{attribute 'GeneratedUsingTerminal: EP3744-0041-0016'}
{attribute addProperty BoxType "EP3744-0041-0016"}
{attribute addProperty Description "EP3744-0041 5Ch. Absolute Pressure 6Ch. Dig. Input 10us 2Ch. Dig. Output 24V 0,5A M8"}
{attribute addProperty Physics "YY"}
{attribute addProperty Id "DIG_InputsAT %I*DIG_Inputs_697E0EF26AI_Inputs_Channel_1AT %I*AI_Inputs_Channel_4521310411AI_Inputs_Channel_2AT %I*AI_Inputs_Channel_4521310411AI_Inputs_Channel_3AT %I*AI_Inputs_Channel_4521310411AI_Inputs_Channel_4AT %I*AI_Inputs_Channel_4521310411DEV_Inputs_DeviceAT %I*DEV_Inputs_Device_5F4E175E5DIG_OutputsAT %Q*DIG_Outputs_DE230DD52DEV_Outputs_DeviceAT %Q*DEV_Outputs_Device_59FFD2471WcStateAT %I*WcState_9091E0EB2InfoDataAT %I*InfoData_32EB74EA10"}
{attribute addProperty CRC "828150484"}
{attribute addProperty Size "70"}
TYPE EP3744_315C92D4 EXTENDS EtcSlaveBoxBase_77A0E4A7 :
STRUCT
	{attribute addProperty Name "DIG_Inputs"}
	DIG_Inputs : DIG_Inputs_697E0EF2;
	{attribute addProperty Name "AI_Inputs_Channel_1"}
	AI_Inputs_Channel_1 : AI_Inputs_Channel_45213104;
	{attribute addProperty Name "AI_Inputs_Channel_2"}
	AI_Inputs_Channel_2 : AI_Inputs_Channel_45213104;
	{attribute addProperty Name "AI_Inputs_Channel_3"}
	AI_Inputs_Channel_3 : AI_Inputs_Channel_45213104;
	{attribute addProperty Name "AI_Inputs_Channel_4"}
	AI_Inputs_Channel_4 : AI_Inputs_Channel_45213104;
	{attribute addProperty Name "DEV_Inputs_Device"}
	DEV_Inputs_Device : DEV_Inputs_Device_5F4E175E;
	{attribute addProperty Name "DIG_Outputs"}
	DIG_Outputs : DIG_Outputs_DE230DD5;
	{attribute addProperty Name "DEV_Outputs_Device"}
	DEV_Outputs_Device : DEV_Outputs_Device_59FFD247;
	{attribute addProperty Name "WcState"}
	WcState : WcState_9091E0EB;
	{attribute addProperty Name "InfoData"}
	InfoData : InfoData_32EB74EA;
END_STRUCT
END_TYPE

(* stored: Version 1.2.0.0, ProductVersion 3.1.4024.9
   DUT EP3744_315C92D4: Id {62da8416-0317-4ab8-9568-44e748466a41} *)
